FUNCTION_BLOCK fbMotion
VAR_INPUT
END_VAR
VAR_OUTPUT
END_VAR
VAR
	MCpower: MC_Power;
	MCStop: MC_Stop;
	McMoveAbs: MC_MoveAbsolute;
	McReset: MC_Reset;
END_VAR

VAR_IN_OUT	
	stAxis	:	ST_Axis;
	axis	:	axis_ref;
END_VAR

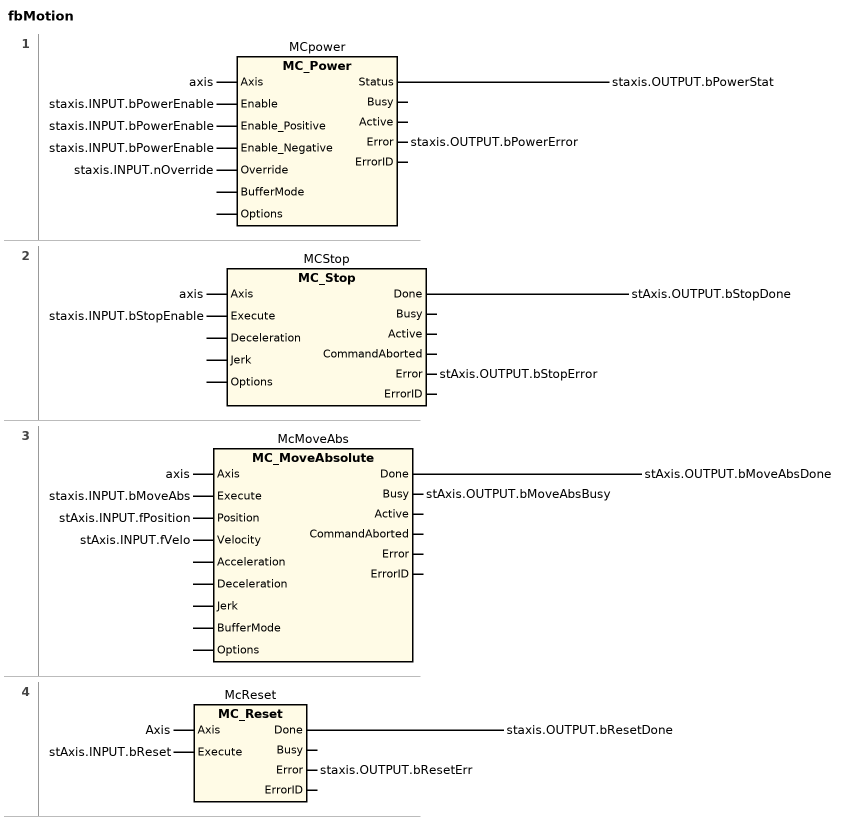
// NETWORK 1
MCpower(
    Axis := axis,
    Enable := staxis.INPUT.bPowerEnable,
    Enable_Positive := staxis.INPUT.bPowerEnable,
    Enable_Negative := staxis.INPUT.bPowerEnable,
    Override := staxis.INPUT.nOverride,
    Error => staxis.OUTPUT.bPowerError); // MC_Power
staxis.OUTPUT.bPowerStat := MCpower.Status;

// NETWORK 2
MCStop(Axis := axis, Execute := staxis.INPUT.bStopEnable, Error => stAxis.OUTPUT.bStopError); // MC_Stop
stAxis.OUTPUT.bStopDone := MCStop.Done;

// NETWORK 3
McMoveAbs(
    Axis := axis,
    Execute := staxis.INPUT.bMoveAbs,
    Position := stAxis.INPUT.fPosition,
    Velocity := stAxis.INPUT.fVelo,
    Busy => stAxis.OUTPUT.bMoveAbsBusy); // MC_MoveAbsolute
stAxis.OUTPUT.bMoveAbsDone := McMoveAbs.Done;

// NETWORK 4
McReset(Axis := Axis, Execute := stAxis.INPUT.bReset, Error => staxis.OUTPUT.bResetErr); // MC_Reset
staxis.OUTPUT.bResetDone := McReset.Done;

END_FUNCTION_BLOCK

(* stored: Version 1.1.0.1, ProductVersion 3.1.4022.18
   POU fbMotion: Id {3827256e-fc14-432e-9323-be08aa701a4e}, SpecialFunc None *)
